// TwinCAT 3 PLC project Factory_Pattern
// ProgramVersion: 3.1.4024.0
// libraries:
//   Tc2_Standard, * (Beckhoff Automation GmbH)
//   Tc2_System, * (Beckhoff Automation GmbH)
//   Tc3_DynamicMemory, * (Beckhoff Automation GmbH)
//   Tc3_Module, * (Beckhoff Automation GmbH)
//   Tc3_UnitTest, * (Zerlauth)
// project tree:
//   Class/ EtherCATDevice.TcPOU, I_EtherCATDevice.TcIO (not stored)
//   Factory/ EtherCATFactory.TcPOU
//   / PlcTask.TcTTO
//   POUs/ MAIN.TcPOU
// real-time tasks:
//   TASK PlcTask: cycle T#10ms, priority 20, ADS port 350
//   TASK PlcTask1: cycle T#10ms, priority 21, ADS port 351
//   TASK PlcTask2: cycle T#10ms, priority 22, ADS port 352
//   TASK PlcTask3: cycle T#10ms, priority 23, ADS port 353
//   TASK PlcTask4: cycle T#10ms, priority 24, ADS port 354
//   TASK PlcTask5: cycle T#10ms, priority 25, ADS port 355
//   TASK PlcTask6: cycle T#10ms, priority 26, ADS port 356
//   TASK PlcTask7: cycle T#10ms, priority 27, ADS port 357
//   TASK PlcTask8: cycle T#10ms, priority 28, ADS port 358
//   TASK PlcTask9: cycle T#10ms, priority 29, ADS port 359
//   TASK PlcTask10: cycle T#10ms, priority 30, ADS port 360
//   TASK PlcTask11: cycle T#10ms, priority 31, ADS port 361

CONFIGURATION Factory_Pattern
    RESOURCE PLC ON TwinCAT3
        TASK PlcTask(INTERVAL := T#10ms, PRIORITY := 20);
        PROGRAM MAIN WITH PlcTask : MAIN;
    END_RESOURCE
END_CONFIGURATION

// ---- POUs/MAIN.TcPOU
PROGRAM MAIN
VAR
	EtherCATIOFactory : EtherCATFactory;
	GetEtherCATDevice: BOOL;
	myDevcie : I_EtherCATDevice;
END_VAR

IF GetEtherCATDevice THEN
	GetEtherCATDevice := FALSE;
	myDevcie := EtherCATIOFactory.CreateEtherCATDevice();
END_IF

END_PROGRAM

// ---- Factory/EtherCATFactory.TcPOU
FUNCTION_BLOCK EtherCATFactory
VAR
	DynamicMemoryManager : FB_DynMem_Manager2;
	DynamicBuffer : FB_DynMem_Buffer(ipMemMan := DynamicMemoryManager);
END_VAR

METHOD PUBLIC CreateEtherCATDevice : I_EtherCATDevice
VAR_INPUT
END_VAR
CreateEtherCATDevice := DynamicMemoryManager.Alloc(nSize := SIZEOF(EtherCATDevice),
													bReset := false);
END_METHOD

END_FUNCTION_BLOCK

// ---- Class/EtherCATDevice.TcPOU
FUNCTION_BLOCK EtherCATDevice IMPLEMENTS I_EtherCATDevice
VAR_INPUT
END_VAR
VAR_OUTPUT
END_VAR
VAR
END_VAR

METHOD IsDeviceOK : BOOL
VAR_INPUT
END_VAR
END_METHOD

END_FUNCTION_BLOCK
